{attribute 'Tc2GvlVarNames'}
VAR_GLOBAL

(*TERMINAL XXXKF1 - EK1100 ******************************************************)


(*TERMINAL 747KF1 - EL4002 ******************************************************)
	qn747KF1_1_LightingIntensityPackAggregationCamera							AT %Q* : INT;
	qn747KF1_2_LightingIntensityPackConfirmationCamera							AT %Q* : INT;

(*TERMINAL 748KF1 - EL4002 ******************************************************)
	qn748KF1_1_LightingIntensityMasterListCamera		AT %Q* : INT;
	qn748KF1_2_Spare										AT %Q* : INT;

(*TERMINAL 763KF1 - EL1008 ******************************************************)
	ib763KF1_1_MasterListCameraTrigSensor					AT %I* : BOOL;
	ib763KF1_5_SpareMasterListCameraTrigSensor			AT %I* : BOOL;		(* Option *)
	ib763KF1_2_AggregationCameraTrigSensor				AT %I* : BOOL;
	ib763KF1_6_SpareAggregationCamera1TrigSensor		AT %I* : BOOL;		(* Option *)
	ib763KF1_3_SpareAggregationCamera2TrigSensor		AT %I* : BOOL;		(* Option *)
	ib763KF1_7_PackQueueIndex								AT %I* : BOOL; 		(* Option *)
	ib763KF1_4_StackQueueIndex								AT %I* : BOOL; 		(* Option *)
	ib763KF1_8_SpareIndex											AT %I* : BOOL;

(*TERMINAL 764KF1 - EL1008 ******************************************************)
	ib764KF1_1_OuterIndexComplete							AT %I* : BOOL;
	ib764KF1_5_SpareCameraTrigSesnor						AT %I* : BOOL;		(* Option *)
	ib764KF1_2_Guard1 										AT %I* : BOOL;		(*FOCKE/GD Master list guard*)
	ib764KF1_6_Guard2										AT %I* : BOOL;		(*FOCKE/GD Master list guard*)
	ib764KF1_3_Guard3 										AT %I* : BOOL;		(*FOCKE/GD Aggregation guard*)
	ib764KF1_7_Guard4 										AT %I* : BOOL;		(*FOCKE/GD Aggregationt guard*)
	ib764KF1_4_OuterBrushOpen								AT %I* : BOOL;
	ib764KF1_8_RejectTowerActive							AT %I* : BOOL;

(*TERMINAL 765KF1 (EL1008 8Ch. Dig. Input 24V, 3ms) ******************************************************)
	ib765KF1_1_FilmInPosition 								AT %I*: BOOL;
	ib765KF1_5_SparePrinterTrigger							AT %I*: BOOL;
	ib765KF1_2_IntermediateCamera1TrigSesnor				AT %I*: BOOL;
	ib765KF1_6_HeatTunelPackReject							AT %I*: BOOL;
	ib765KF1_3_OuterAtAdditionalConveyor01 				AT %I*: BOOL;
	ib765KF1_7_IntermediateCamera2TrigSesnor				AT %I*: BOOL;
	ib765KF1_4_OuterAtReject									AT %I*: BOOL;		(*AdditionalConveyor01*)
	ib765KF1_8_RejectConfirmation	 						AT %I*: BOOL;		(*AdditionalConveyor01*)

(*TERMINAL 766KF1 - EL1008 ******************************************************)
	ib766KF1_1_RejectCylinderExtended						AT %I* : BOOL;
	ib766KF1_5_RejectCylinderRetracted						AT %I* : BOOL;		(*  *)
	ib766KF1_2_RejectBinFull 									AT %I* : BOOL;		(*AdditionalConveyor01*)
	ib766KF1_6_ExitBlockedAdditionalConveyor01				AT %I* : BOOL;
	ib766KF1_3_IntermediateCamera3TrigSesnor				AT %I* : BOOL;
	ib766KF1_7_Spare											AT %I* : BOOL;	(*Potentially for GD Additional Master list guard*)
	ib766KF1_4_Spare											AT %I* : BOOL;		(* Guard5 Potentially for GD Wrapper door*)
	ib766KF1_8_Spare											AT %I* : BOOL;			(* Guard6 Potentially for GD Wrapper door*)

(*TERMINAL 767KF1 - EL1008 ******************************************************)
	ib767KF1_1_ConveyorInterfaceInputSignal1				AT %I* : BOOL;
	ib767KF1_5_ConveyorInterfaceInputSignal2				AT %I* : BOOL;		(*  *)
	ib767KF1_2_RejectTower2Active							AT %I* : BOOL;		(**)
	ib767KF1_6_Spare											AT %I* : BOOL;
	ib767KF1_3_Spare											AT %I* : BOOL;
	ib767KF1_7_Spare 											AT %I* : BOOL;
	ib767KF1_4_Spare											AT %I* : BOOL;
	ib767KF1_8_Spare											AT %I* : BOOL;


(*TERMINAL 783KF1 - EL2008 ******************************************************)
	qb783KF1_1_MasterListCameraPower						AT %Q* : BOOL;
	qb783KF1_5_SpareMasterListCameraPower					AT %Q* : BOOL;	(* Option *)
	qb783KF1_2_SpareAggregationCameraPower				AT %Q* : BOOL;	(* Option *)
	qb783KF1_6_AggregationCamera1Power					AT %Q* : BOOL;
	qb783KF1_3_AggregationCamera2Power					AT %Q* : BOOL;
	qb783KF1_7_ConfirmationCamera1Power					AT %Q* : BOOL; 	(* Option *)
	qb783KF1_4_ConfirmationCamera2Power					AT %Q* : BOOL; 	(* Option *)
	qb783KF1_8_PLCControlledAggCamerasLightning			AT %Q* : BOOL;

(*TERMINAL 784KF1 - EL2008 ******************************************************)
	qb784KF1_1_MasterListCameraTrigger						AT %Q* : BOOL;
	qb784KF1_5_SpareMasterListCameraTrigger				AT %Q* : BOOL;	(* Option *)
	qb784KF1_2_AggregationCameraTrigger					AT %Q* : BOOL;
	qb784KF1_6_SpareAggregationCamera1Trigger			AT %Q* : BOOL; 	(* Option *)
	qb784KF1_3_SpareAggregationCamera2Trigger			AT %Q* : BOOL; 	(* Option *)
	qb784KF1_7_ConfirmationCamera1Trigger					AT %Q* : BOOL; 	(* Option *)
	qb784KF1_4_ConfirmationCamera2Trigger					AT %Q* : BOOL; 	(* Option *)
	qb784KF1_8_PLCControlledConfCameraLightning			AT %Q* : BOOL;

(*TERMINAL 785KF1 (EL2008 8Ch. Dig. Output 24V, 3ms) ******************************************************)
	qb785KF1_1_IntermediateCamera1Trigger					AT %Q*: BOOL;
	qb785KF1_5_IntermediateCamera1Power					AT %Q*: BOOL;
	qb785KF1_2_IntermediateCamera2Trigger					AT %Q*: BOOL;
	qb785KF1_6_IntermediateCamera3Power					AT %Q*: BOOL;
	qb785KF1_3_RejectCylinderExtended						AT %Q*: BOOL;			(*AdditionalConveyor01*)
	qb785KF1_7_RjectCylinderRetracted						AT %Q*: BOOL;			(*AdditionalConveyor01*)
	qb785KF1_4_IntermediateCamera3Trigger					AT %Q*: BOOL;
	qb785KF1_8_IntermediateCamera3Power					AT %Q*: BOOL;

(*TERMINAL 786KF1 - EL2008 ******************************************************)
	qb786KF1_1_ConveyorInterfaceOutputSignal1				AT %Q* : BOOL;
	qb786KF1_5_ConveyorInterfaceOutputSignal2				AT %Q* : BOOL;	(* Option *)
	qb786KF1_2_Spare											AT %Q* : BOOL;	(* Option *)
	qb786KF1_6_Spare											AT %Q* : BOOL;
	qb786KF1_3_Spare											AT %Q* : BOOL;
	qb786KF1_7_Spare											AT %Q* : BOOL; 	(* Option *)
	qb786KF1_4_Spare											AT %Q* : BOOL; 	(* Option *)
	qb786KF1_8_PLCControlledMLCamerasLightning			AT %Q* : BOOL;

END_VAR

(* stored: Version 1.1.0.1, ProductVersion 3.1.4024.15
   GVL IOVariablesPLAS_OC: Id {c4c048eb-982e-4c5b-a6a5-5deb348a3110} *)
